// TIA Portal V18 export
// export: Created 2026-01-09T11:23:37.6258747Z, ExportSetting WithDefaults, DisplayName Totally Integrated Automation Portal, DisplayVersion V18 Update 5, DisplayName TIA Portal Openness, DisplayVersion V18 Update 5, DisplayName TIA Portal Teamcenter Gateway, DisplayVersion V18, DisplayName TIA Portal Version Control Interface, DisplayVersion V18, DisplayName SINAMICS Startdrive Advanced, DisplayVersion V18 SP2 Update 1, DisplayName SINAMICS Startdrive G110M, G120, G120C, G120D, G120P, G115D, DisplayVersion V18 SP2 Update 1, DisplayName SINAMICS Startdrive G130, G150, S120, S150, SINAMICS MV, S210, G220, S200, DisplayVersion V18 SP2 Update 1, DisplayName STEP 7 Professional, DisplayVersion V18 Update 5, DisplayName STEP 7 Safety, DisplayVersion V18, DisplayName WinCC Professional, DisplayVersion V18 Update 5
Screen "310History"  1280x800, Number=310, Template=T1
  ScreenLayer "Layer_0"
    Button "按钮_7" at 256,725 size 128x75  Mode=Text, PictureOff=向左箭头_0, StyleItem=BtnActive20, TextOff="历史报警 / Alarm history / Alarm História"
      on Click: ActivateScreen(Screen name := , Object number := 0); SetTag(Tag := Sys_VersionManagement_HMIPageID, Value := 310)
    Button "按钮_1" at 128,725 size 128x75  Mode=Text, PictureOff=向左箭头_0, StyleItem=BtnNormal20, TextOff="当前报警 / Alarm"
      on Click: ActivateScreen(Screen name := 300Main, Object number := 0); SetTag(Tag := Sys_VersionManagement_HMIPageID, Value := 300)
